(* IEC 61131-3 sources: RL_MAR/experiments/comparison/autoplc/results/deepseek-ai-DeepSeek-V3.2_20260508_111905/med_26, 1 file *)

(* ---- med_26_1.st ---- *)
FUNCTION_BLOCK BookSorting
VAR_INPUT
    RFID1 : BOOL;
    RFID2 : BOOL;
    RFID3 : BOOL;
END_VAR

VAR_OUTPUT
    Motor : BOOL;
    Bin1 : BOOL;
    Bin2 : BOOL;
    Bin3 : BOOL;
END_VAR

VAR
    // Internal variables for processing
    AnyRFIDDetected : BOOL;
END_VAR

// Main control logic
AnyRFIDDetected := RFID1 OR RFID2 OR RFID3;

// Control motor based on RFID detection
IF AnyRFIDDetected THEN
    Motor := TRUE;

    // Determine which bin to open with priority: RFID1 > RFID2 > RFID3
    IF RFID1 THEN
        Bin1 := TRUE;
        Bin2 := FALSE;
        Bin3 := FALSE;
    ELSIF RFID2 THEN
        Bin1 := FALSE;
        Bin2 := TRUE;
        Bin3 := FALSE;
    ELSIF RFID3 THEN
        Bin1 := FALSE;
        Bin2 := FALSE;
        Bin3 := TRUE;
    ELSE
        // Safety fallback - should not reach here if AnyRFIDDetected is TRUE
        Bin1 := FALSE;
        Bin2 := FALSE;
        Bin3 := FALSE;
    END_IF;
ELSE
    // No RFID detection - stop motor and close all bins
    Motor := FALSE;
    Bin1 := FALSE;
    Bin2 := FALSE;
    Bin3 := FALSE;
END_IF;

END_FUNCTION_BLOCK
